// SIMATIC STEP 7 (V5.x) project S_Modos
// CPU: CPU312(1)
// station: P_ADR_BUS
// station: Hardware
// station: Equipo SIMATIC 300
// program: Programa S7(1)

SYMBOL_TABLE
"Global"	DB 1	DB 1
"Modo1"	DB 2	DB 2
"Modo2"	DB 3	DB 3
"MODOS"	FC 3	FC 3
"MODO_1"	I 124.0	BOOL
"MODO_2"	I 124.1	BOOL
"BIT_DE_TRABAJO"	I 124.2	BOOL
"Cycle Execution"	OB 1	OB 1
"PLANCHAS_GL"	PIW 651	WORD
"STBY"	Q 100.0	BOOL
END_SYMBOL_TABLE

FUNCTION "MODOS" : VOID	// FC 3
VERSION : 0.1
VAR_INPUT
  BIT_DE_TRABAJO : BOOL ;
  MODO1 : BOOL ;
  MODO2 : BOOL ;
END_VAR
VAR_OUTPUT
  STBY : BOOL ;
END_VAR
VAR_TEMP
  X60 : BOOL ;
  X61 : BOOL ;
  X62 : BOOL ;
  FP_BDT : BOOL ;
  FP_X61 : BOOL ;
  FP_X62 : BOOL ;
END_VAR
BEGIN
NETWORK
TITLE =
      A     #BIT_DE_TRABAJO;
      FP    #FP_BDT;
      S     #X60;
      R     #X61;
      R     #X62;
NETWORK
TITLE =
      A     #X60;
      A     #MODO1;
      R     #X60;
      S     #X61;
NETWORK
TITLE =
      A     #X60;
      A     #MODO2;
      R     #X60;
      S     #X62;
NETWORK
TITLE =
      A     #X61;
      AN    #MODO1;
      R     #X61;
      S     #X60;
NETWORK
TITLE =
      A     #X62;
      AN    #MODO2;
      R     #X62;
      S     #X60;
NETWORK
TITLE =
      A     #X60;
      =     #STBY;
NETWORK
TITLE = Numero de planchas por bobina y peso Modo 1
      A     #X61;
      JCN   _001;
      L     "Modo1".PLANCHAS;
      T     "Global".PLANCHAS;
      L     "Modo1".PESO_PAELLERA;
      T     "Global".PESO_PAELLERA;
      L     "Modo1".PESO_WOK;
      T     "Global".PESO_WOK;
      L     "Modo1".PESO_SARTEN;
      T     "Global".PESO_SARTEN;
      L     "Modo1".PESO_CACEROLA;
      T     "Global".PESO_CACEROLA;
_001: NOP   0;
NETWORK
TITLE =
      A     #X62;
      JCN   _002;
      L     "Modo2".PLANCHAS;
      T     "Global".PLANCHAS;
      L     "Modo2".PESO_PAELLERA;
      T     "Global".PESO_PAELLERA;
      L     "Modo2".PESO_WOK;
      T     "Global".PESO_WOK;
      L     "Modo2".PESO_SARTEN;
      T     "Global".PESO_SARTEN;
      L     "Modo2".PESO_CACEROLA;
      T     "Global".PESO_CACEROLA;
_002: NOP   0;
END_FUNCTION

DATA_BLOCK "Global"	// DB 1
VERSION : 0.1
  STRUCT
   PESO_CACEROLA : REAL ;	//Peso Bobina Cacerolas
   PESO_WOK : REAL ;	//Peso Bobina Wok
   PESO_SARTEN : REAL ;	//Peso Bobina Sarten
   PESO_PAELLERA : REAL ;	//Peso Bobina Paellera
   PLANCHAS : WORD ;	//Número de planchas por bobina
  END_STRUCT ;	
BEGIN
   PESO_CACEROLA := 1.000000e+02;
   PESO_WOK := 1.100000e+02;
   PESO_SARTEN := 1.200000e+02;
   PESO_PAELLERA := 1.300000e+02;
   PLANCHAS := W#16#100;
END_DATA_BLOCK

DATA_BLOCK "Modo1"	// DB 2
VERSION : 0.1
  STRUCT
   PESO_CACEROLA : REAL  := 1.000000e+002;	//Peso Bobina Cacerolas
   PESO_WOK : REAL  := 1.100000e+002;	//Peso Bobina Wok
   PESO_SARTEN : REAL  := 1.200000e+002;	//Peso Bobina Sarten
   PESO_PAELLERA : REAL  := 1.300000e+002;	//Peso Bobina Paellera
   PLANCHAS : WORD  := W#16#100;	//Número de planchas por bobina
  END_STRUCT ;	
BEGIN
   PESO_CACEROLA := 1.000000e+02;
   PESO_WOK := 1.100000e+02;
   PESO_SARTEN := 1.200000e+02;
   PESO_PAELLERA := 1.300000e+02;
   PLANCHAS := W#16#100;
END_DATA_BLOCK

DATA_BLOCK "Modo2"	// DB 3
VERSION : 0.1
  STRUCT
   PESO_CACEROLA : REAL  := 2.000000e+002;	//Peso Bobina Cacerolas
   PESO_WOK : REAL  := 2.200000e+002;	//Peso Bobina Wok
   PESO_SARTEN : REAL  := 2.400000e+002;	//Peso Bobina Sarten
   PESO_PAELLERA : REAL  := 2.600000e+002;	//Peso Bobina Paellera
   PLANCHAS : WORD  := W#16#200;	//Número de planchas por bobina
  END_STRUCT ;	
BEGIN
   PESO_CACEROLA := 2.000000e+02;
   PESO_WOK := 2.200000e+02;
   PESO_SARTEN := 2.400000e+02;
   PESO_PAELLERA := 2.600000e+02;
   PLANCHAS := W#16#200;
END_DATA_BLOCK

ORGANIZATION_BLOCK "Cycle Execution"	// OB 1
TITLE = "Main Program Sweep (Cycle)"
VERSION : 0.1
VAR_TEMP
  OB1_EV_CLASS : BYTE ;	//Bits 0-3 = 1 (Coming event), Bits 4-7 = 1 (Event class 1)
  OB1_SCAN_1 : BYTE ;	//1 (Cold restart scan 1 of OB 1), 3 (Scan 2-n of OB 1)
  OB1_PRIORITY : BYTE ;	//Priority of OB Execution
  OB1_OB_NUMBR : BYTE ;	//1 (Organization block 1, OB1)
  OB1_RESERVED_1 : BYTE ;	//Reserved for system
  OB1_RESERVED_2 : BYTE ;	//Reserved for system
  OB1_PREV_CYCLE : INT ;	//Cycle time of previous OB1 scan (milliseconds)
  OB1_MIN_CYCLE : INT ;	//Minimum cycle time of OB1 (milliseconds)
  OB1_MAX_CYCLE : INT ;	//Maximum cycle time of OB1 (milliseconds)
  OB1_DATE_TIME : DATE_AND_TIME ;	//Date and time OB1 started
END_VAR
BEGIN
NETWORK
TITLE =
      SET;
      CALL  "MODOS" (
           BIT_DE_TRABAJO           := "BIT_DE_TRABAJO",
           MODO1                    := "MODO_1",
           MODO2                    := "MODO_2",
           STBY                     := "STBY");
END_ORGANIZATION_BLOCK
